(* Schneider Machine Expert - Basic project FirstTest, file version 3.0.0.0 *)
(* ProjectInformations: Name=t-New project *)

HARDWARE
  Cpu 0: TM221CE16R
  ModuleExtensionObject 0: TM3DQ16R/G
  EthernetConfiguration: NetworkName=M221, IpAllocationMode=FixedAddress, IpAddress=0.0.0.0, SubnetMask=0.0.0.0
  SerialLineConfiguration: Baud=Baud19200, Parity=ParityEven, DataBits=DataBits8, StopBits=StopBits1, PhysicalMedium=PhysicalMediumRs485, TransmissionMode=TransmissionModeModbusRtu, SlaveId=1, Addressing=SlaveAddressing
  MastTask: UsePeriodScanMode=false, PeriodScan=100
  FastTask: Period=255
  CpuBehavior: StartingMode=StartAsPreviousState, AutoSaveRamOnEeprom=true, WatchdogPeriod=250

SYMBOLS  (address, symbol, comment, settings)
  %M0       SENSOR_CAPACITIVO  "ON = hay líquido. Si está invertido, cambiar a contacto NC aquí"
  %M1       MOLDE_DET  "ON = molde detectado. Si sale Light-ON, cambiar a NC en Rung 2"
  %M10      RESET_SW  "Reset de falla por software (forzar 1 y regresar a 0)"
  %S6       SB_TB1S  "Time base of 1 s generated by an internal clock"
  %S13      SB_FIRSTRUN  "Indicates the first controller cycle in RUN mode"
  %MW0      ESTADO  "Estado FSM: 0 = ESPERA, 1 = LLENANDO, 2 = FALLA"
  %TM0      T_NIVEL_BAJO  "Nivel bajo continuo 2 s antes de llenar"  [Preset=2, Base=OneSecond]
  %TM1      T_MOLDES  "Mantiene "hay moldes" 5 s después del último"  [Type=TOF, Preset=5, Base=OneSecond]
  %TM2      T_TIMEOUT  "Tiempo máximo de llenado → FALLA"  [Preset=30, Base=OneSecond]
  %TM3      T_REPOSO  "Reposo en ESPERA antes de volver a llenar"  [Preset=5, Base=OneSecond]
  %I0.0     CAP_NIVEL  "Capacitivo Autonics CR18 - ON = hay líquido"
  %I0.1     FOTO_MOLD  "Fotoeléctrico E3F-20DC1 vía relé K2"
  %I0.2     BTN_RESET  "Pulsador NA de reset de falla (opcional)"
  %Q1.0     EV_LLENADO  "Relé K1 → electroválvula de llenado"
  %Q1.1     LAMP_FALLA  "Lámpara de falla (parpadea en FALLA)"

POU Latex pools
  (* SectionNumber=1 *)

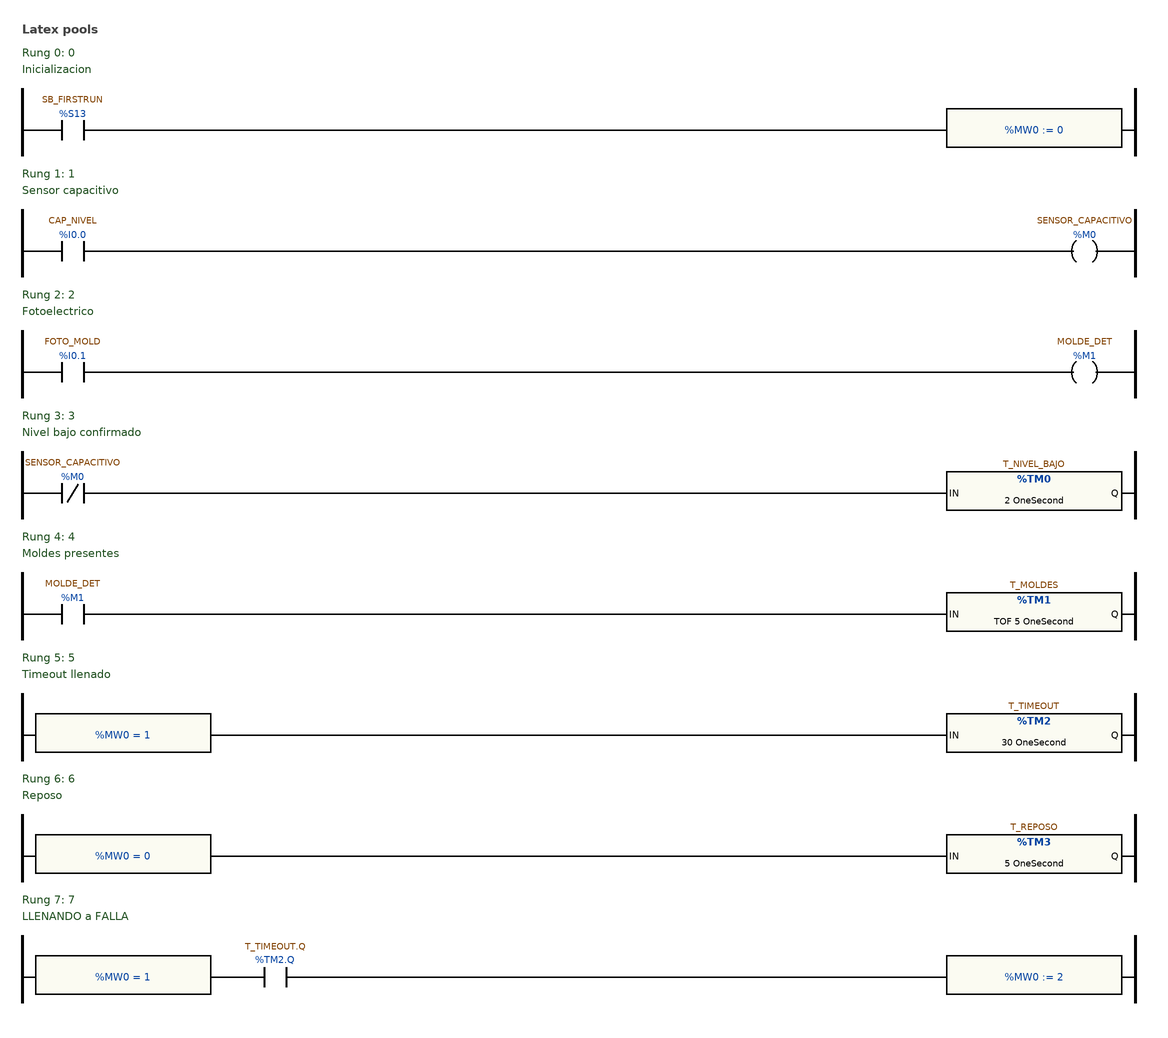

// Rung 0: 0
// Inicializacion
  LD %S13                 (* SB_FIRSTRUN *)
  [ %MW0 := 0 ]           (* ESTADO *)
  // as ST:
  //   IF SB_FIRSTRUN THEN ESTADO := 0; END_IF;

// Rung 1: 1
// Sensor capacitivo
  LD %I0.0                (* CAP_NIVEL *)
  ST %M0                  (* SENSOR_CAPACITIVO *)
  // as ST:
  //   SENSOR_CAPACITIVO := CAP_NIVEL;

// Rung 2: 2
// Fotoelectrico
  LD %I0.1                (* FOTO_MOLD *)
  ST %M1                  (* MOLDE_DET *)
  // as ST:
  //   MOLDE_DET := FOTO_MOLD;

// Rung 3: 3
// Nivel bajo confirmado
  BLK %TM0                (* T_NIVEL_BAJO *)
  LDN %M0                 (* SENSOR_CAPACITIVO *)
  IN
  END_BLK
  // as ST:
  //   T_NIVEL_BAJO(IN := NOT SENSOR_CAPACITIVO);

// Rung 4: 4
// Moldes presentes
  BLK %TM1                (* T_MOLDES *)
  LD %M1                  (* MOLDE_DET *)
  IN
  END_BLK
  // as ST:
  //   T_MOLDES(IN := MOLDE_DET);

// Rung 5: 5
// Timeout llenado
  BLK %TM2                (* T_TIMEOUT *)
  LD [ %MW0 = 1 ]         (* ESTADO *)
  IN
  END_BLK
  // as ST:
  //   T_TIMEOUT(IN := ESTADO = 1);

// Rung 6: 6
// Reposo
  BLK %TM3                (* T_REPOSO *)
  LD [ %MW0 = 0 ]         (* ESTADO *)
  IN
  END_BLK
  // as ST:
  //   T_REPOSO(IN := ESTADO = 0);

// Rung 7: 7
// LLENANDO a FALLA
  LD [ %MW0 = 1 ]         (* ESTADO *)
  AND %TM2.Q              (* T_TIMEOUT *)
  [ %MW0 := 2 ]           (* ESTADO *)
  // as ST:
  //   IF ESTADO = 1 AND T_TIMEOUT.Q THEN ESTADO := 2; END_IF;

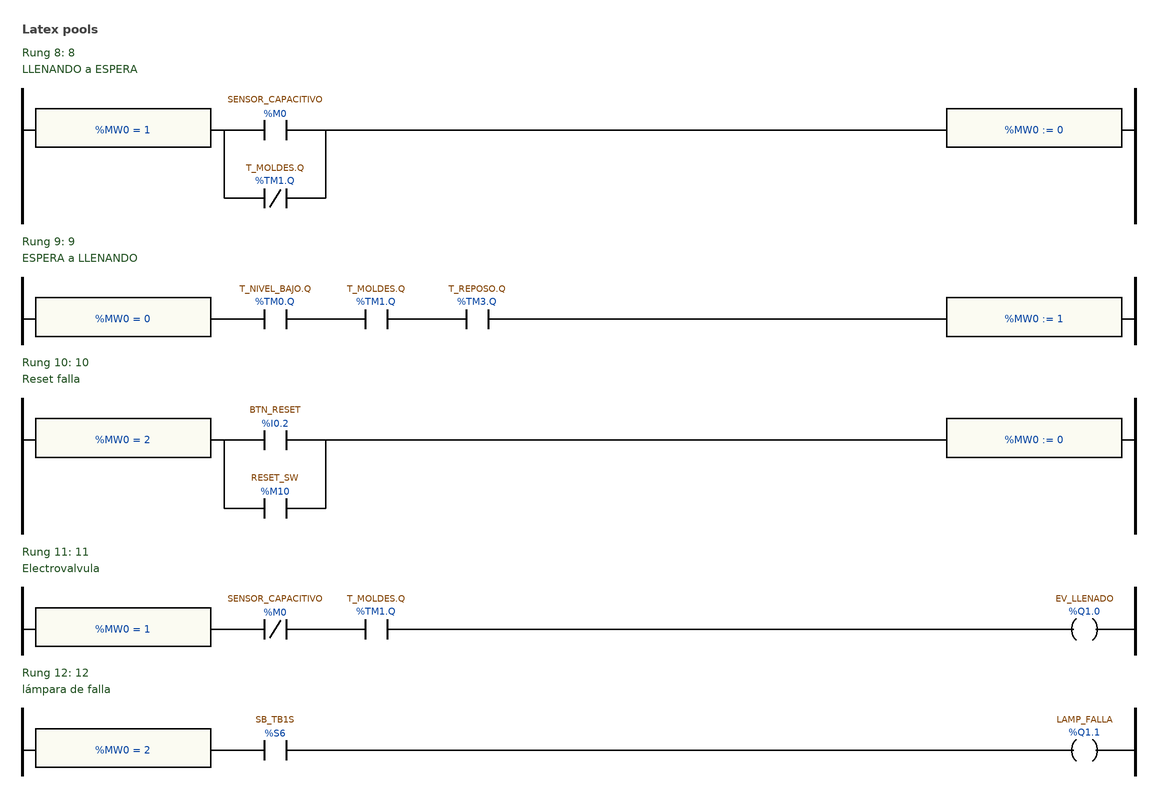

// Rung 8: 8
// LLENANDO a ESPERA
  LD [ %MW0 = 1 ]         (* ESTADO *)
  AND( %M0                (* SENSOR_CAPACITIVO *)
  ORN %TM1.Q              (* T_MOLDES *)
  )
  [ %MW0 := 0 ]           (* ESTADO *)
  // as ST:
  //   IF ESTADO = 1 AND (SENSOR_CAPACITIVO OR NOT T_MOLDES.Q) THEN ESTADO := 0; END_IF;

// Rung 9: 9
// ESPERA a LLENANDO
  LD [ %MW0 = 0 ]         (* ESTADO *)
  AND %TM0.Q              (* T_NIVEL_BAJO *)
  AND %TM1.Q              (* T_MOLDES *)
  AND %TM3.Q              (* T_REPOSO *)
  [ %MW0 := 1 ]           (* ESTADO *)
  // as ST:
  //   IF ESTADO = 0 AND T_NIVEL_BAJO.Q AND T_MOLDES.Q AND T_REPOSO.Q THEN ESTADO := 1; END_IF;

// Rung 10: 10
// Reset falla
  LD [ %MW0 = 2 ]         (* ESTADO *)
  AND( %I0.2              (* BTN_RESET *)
  OR %M10                 (* RESET_SW *)
  )
  [ %MW0 := 0 ]           (* ESTADO *)
  // as ST:
  //   IF ESTADO = 2 AND (BTN_RESET OR RESET_SW) THEN ESTADO := 0; END_IF;

// Rung 11: 11
// Electrovalvula
  LD [ %MW0 = 1 ]         (* ESTADO *)
  ANDN %M0                (* SENSOR_CAPACITIVO *)
  AND %TM1.Q              (* T_MOLDES *)
  ST %Q1.0                (* EV_LLENADO *)
  // as ST:
  //   EV_LLENADO := ESTADO = 1 AND NOT SENSOR_CAPACITIVO AND T_MOLDES.Q;

// Rung 12: 12
// lámpara de falla
  LD [ %MW0 = 2 ]         (* ESTADO *)
  AND %S6                 (* SB_TB1S *)
  ST %Q1.1                (* LAMP_FALLA *)
  // as ST:
  //   LAMP_FALLA := ESTADO = 2 AND SB_TB1S;
